FUNCTION_BLOCK F_INT_AS_STRING (* Convert INT to STRING *)
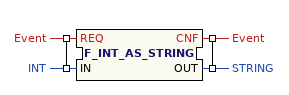
  EVENT_INPUT
    REQ WITH IN; (* Normal Execution Request *)
  END_EVENT
  EVENT_OUTPUT
    CNF WITH OUT; (* Execution Confirmation *)
  END_EVENT
  VAR_INPUT
    IN : INT;
  END_VAR
  VAR_OUTPUT
    OUT : STRING;
  END_VAR
END_FUNCTION_BLOCK
